{attribute 'linkalways'} 
{attribute 'no_explicit_call' := 'This FB is a CLASS and must be accessed using methods or properties'}
{attribute 'enable_dynamic_creation'}
FUNCTION_BLOCK Node_F_VN_ApplyYAxisInversionToAffineTransformation EXTENDS VisionNode
VAR
    aTransformationMatrix : _TcVnMatrix2x3_LREAL;
    hrPrev : _HRESULT(S_OK);
	hresult : _HRESULT(S_OK);
END_VAR

METHOD PUBLIC  Clone : I_Node
VAR
	pNode : POINTER TO Node_F_VN_ApplyYAxisInversionToAffineTransformation;
END_VAR
pNode := __NEW(Node_F_VN_ApplyYAxisInversionToAffineTransformation);
Clone := pNode^;
END_METHOD

METHOD FB_init : BOOL
VAR_INPUT
	bInitRetains : BOOL; // if TRUE, the retain variables are initialized (warm start / cold start)
	bInCopyCode : BOOL;  // if TRUE, the instance afterwards gets moved into the copy code (online change)
END_VAR
AddInput('aTransformationMatrix', aTransformationMatrix);
AddInput('hrPrev', hrPrev);
AddOutput('aTransformationMatrix', aTransformationMatrix);
AddOutput('hresult',hresult);
END_METHOD

METHOD PROTECTED OnExecute : HRESULT
hresult.Value := F_VN_ApplyYAxisInversionToAffineTransformation(
    aTransformationMatrix := aTransformationMatrix.Value,
	hrPrev:= hrPrev.Value);
END_METHOD

METHOD PUBLIC PreExecutionCheck
VAR_INPUT
	Check : I_PreExecutionChecks;
END_VAR
END_METHOD

END_FUNCTION_BLOCK

(* stored: Version 1.1.0.1, ProductVersion 3.1.4024.13
   POU Node_F_VN_ApplyYAxisInversionToAffineTransformation: Id {6caaa8e9-a519-0756-2d5d-ea2123737f6a}, SpecialFunc None
   Folder Constructor: Id {1759388d-dd66-0ba0-3715-c8fccedcd110}
   Method Clone: Id {7e5c0816-5d74-004c-1aa0-f5bc65678149}
   Method FB_init: Id {d6afebcb-1a47-0016-3ef9-0811ae509ddf}
   Method OnExecute: Id {ff234316-1f9b-00e0-092d-7557ec733d19}
   Method PreExecutionCheck: Id {95091361-6145-0e86-2eed-64d95c770b17} *)
